// TIA Portal V19 export
DATA_BLOCK "Boiler_2"   // DB12
// stored: InstanceOfName BoilerAlarm, InstanceOfType FB
"BoilerAlarm"
   // VAR_INPUT
   //    "Alarm Bit" : Bool;
   // END_VAR
   // VAR
   //    Boiler : Program_Alarm;
   // END_VAR
BEGIN
END_DATA_BLOCK
